FUNCTION fPlatformAngleTheta1 : LREAL
VAR_INPUT
	fStroke : LREAL;
END_VAR
VAR
	fAngleBeta		: LREAL;
	fCylinderLength	: LREAL;
	fMinLength 		: LREAL; 
END_VAR

fMinLength := G_StablePlatformParameters.fMinLengthPlatformCylinder;

fCylinderLength := fStroke + fMinLength;

fAngleBeta := ACOS((G_StablePlatformParameters.fLengthA*G_StablePlatformParameters.fLengthA +  G_StablePlatformParameters.fLengthC*G_StablePlatformParameters.fLengthC - fCylinderLength*fCylinderLength) / (2 * G_StablePlatformParameters.fLengthA * G_StablePlatformParameters.fLengthC));

fPlatformAngleTheta1 := -(fAngleBeta - G_StablePlatformParameters.fOffsetAngleRad);

END_FUNCTION

(* stored: Version 1.1.0.1, ProductVersion 3.1.4024.12
   POU fPlatformAngleTheta1: Id {4ff9792d-777c-4893-b06a-b7f302f2ee5a}, SpecialFunc None *)
